// TIA Portal project "PLC-Lab-Projektvorlage-1500-Advanced-V13-PlcLabEdit" (V13)

(* hardware
DEVICE "S71500/ET200MP-Station_1"  S7-1500 station
   slot 0: "Profilschiene_0"  6ES7 590-1***0-0AA0
   slot 0: "PS 25W 24VDC_1"  PS 25W 24VDC  6ES7 505-0KA00-0AB0  V1.0
   slot 1: "PLC_PlcLabProjektVorlage"  CPU 1511-1 PN  6ES7 511-1AK00-0AB0  V1.8
   slot 2: "AI 8xU/I/RTD/TC ST_1"  AI 8xU/I/RTD/TC ST  6ES7 531-7KF00-0AB0  V2.0
   slot 3: "DI 16x24VDC BA_1"  DI 16x24VDC BA  6ES7 521-1BH10-0AA0  V1.0
*)

// ===== PLC "PLC_PlcLabProjektVorlage"  CPU 1511-1 PN =====

FUNCTION "MHJ-PLC-Lab-Function-S71500" : Void   // FC1, SCL
{ S7_Optimized_Access := 'FALSE' }
VERSION : 0.1
BEGIN

   #Value:=PEEK(area := 16#82,
        dbNumber := 0,
        byteOffset := 511);
   #Value := #Value + 1;

   POKE(area := 16#82,
        dbNumber := 0,
        byteOffset := 511,
        value := #Value);

   POKE(area := 16#82,
        dbNumber := 0,
        byteOffset := 1016,
        value := #Value_01_DW);
   POKE(area := 16#82,
        dbNumber := 0,
        byteOffset := 1020,
        value := #Value_02_DW);

   #MaxDiByteTemp := 462;
   IF #MaxDiByte < 463 THEN
       #MaxDiByteTemp := #MaxDiByte;
   END_IF;

   #MinDiByteTemp := 0;
   IF #MaxDiByteTemp >= #MinDiByte & #MinDiByte >= 0 THEN
       #MinDiByteTemp := #MinDiByte;
   END_IF;

   FOR #ForCounter := #MinDiByteTemp TO #MaxDiByteTemp DO
       #Value := PEEK(area := 16#1,
                      dbNumber := 0,
                      byteOffset := #ForCounter);
       POKE(area := 16#81,
            dbNumber := 0,
            byteOffset := #ForCounter,
            value := #Value);
   END_FOR;

   #Value := PEEK(area := 16#1,
                  dbNumber := 0,
                  byteOffset := 512);
   POKE(area := 16#82,
        dbNumber := 0,
        byteOffset := 512,
        value := #Value);
END_FUNCTION

FUNCTION "MHJ-PLC-Lab-Function-S71500-NextInputArea" : Void   // FC2, SCL
{ S7_Optimized_Access := 'FALSE' }
VERSION : 0.1
BEGIN


   #MaxDiByteTemp := -1;
   IF #MaxDiByte < 463 THEN
       #MaxDiByteTemp := #MaxDiByte;
   END_IF;

   #MinDiByteTemp := -1;
   IF #MaxDiByteTemp >= #MinDiByte & #MinDiByte >= 0 THEN
       #MinDiByteTemp := #MinDiByte;
   END_IF;

   IF #MaxDiByteTemp >= 0 & #MinDiByte >= 0 THEN
       FOR #ForCounter := #MinDiByteTemp TO #MaxDiByteTemp DO
           #Value := PEEK(area := 16#1,
                          dbNumber := 0,
                          byteOffset := #ForCounter);
           POKE(area := 16#81,
                dbNumber := 0,
                byteOffset := #ForCounter,
                value := #Value);
       END_FOR;

   END_IF;
END_FUNCTION

ORGANIZATION_BLOCK "Main"   // OB1, FBD, ProgramCycle
TITLE = "Main Program Sweep (Cycle)"
{ S7_Optimized_Access := 'FALSE' }
VERSION : 0.1
   VAR_TEMP   // added for the SCL form of the ladder/FBD networks
      _w1 : Bool;
      _w2 : Bool;
   END_VAR
BEGIN

REGION Network 1
   // MinDiByte: Die minimale Byteadresse der in PLC-Lab verwendbaren Eingänge.
   // MaxDiByte: Die maximale Byteadresse der in PLC-Lab verwendbaren Eingänge.
   // 
   // Bei den folgenden Aufrufen können die Eingangsbytes 0 bis 15 in PLC-Lab verwendet werden. 
   // Sind weitere Eingangsbereiche notwendig, dann können zusätzliche "MHJ-PLC-Lab-Function-S71500-NextInputArea" aufgerufen werden.
   // 
   // Vorgehensweise wenn mehr Bytes oder andere Eingangsadressen zu verwenden sind:
   // 1. Platzieren der Eingangsbaugruppen in der Hardwarekonfiguration.
   // 2. Prozessabbild der Module auf "Keiner" einstellen, deren Eingänge von PLC-Lab beeinflusst werden sollen.
   // 3. Angabe der gewünschten Eingangs-Byteadressen an MinDiByte und MaxDiByte.
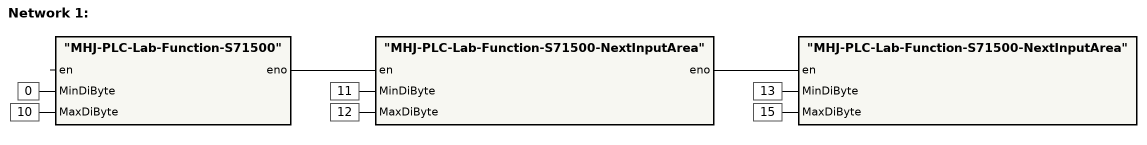
   "MHJ-PLC-Lab-Function-S71500"(MinDiByte := 0, MaxDiByte := 10, ENO => #_w1);
   "MHJ-PLC-Lab-Function-S71500-NextInputArea"(EN := #_w1, MinDiByte := 11, MaxDiByte := 12, ENO => #_w2);
   IF #_w2 THEN "MHJ-PLC-Lab-Function-S71500-NextInputArea"(MinDiByte := 13, MaxDiByte := 15); END_IF;
END_REGION
END_ORGANIZATION_BLOCK